Staubli VAL3: hmns.pgx

public program hmns(num x_nSec, num& x_nHour[], num& x_nMinute[], num& x_nSecond[])
begin
  //-----------------------------------------------------------------------
  //Header begin
  //Description of program
  //  Decompose num seconds in num Hours,minutes, seconds.
  //
  //Input parameters
  //  num x_nSec :
  //    role : put a numerical expression that you want to convert in Hmns
  //
  //Output parameters
  //  num x_nHour :
  //    role : numerical expression that contains Hours
  //  num x_nMinute :
  //    role : numerical expression that contains Minutes
  //  num x_nSecond :
  //    role : numerical expression that contains Seconds
  //
  //Example
  //  call hmns(54200,l_nHour,l_nMinute,l_nSecond)
  //
  //History
  //  Creation : 28-04-08 - f.Rob
  //Header end
  //-----------------------------------------------------------------------
  x_nHour=roundDown(x_nSec/3600)
  x_nMinute=roundDown((x_nSec%3600)/60)
  x_nSecond=roundDown(x_nSec-x_nHour*3600-x_nMinute*60)
end
